FUNCTION setOutInt : INT
VAR_INPUT
	bol_GlobalEnableForce: BOOL;
	p_Output: POINTER TO T_Ctrl_IoInt;
END_VAR

// Copy real values
p_Output^.state := p_Output^.intern;

IF (p_Output^.EnForce AND bol_GlobalEnableForce) THEN
	p_Output^.map := p_Output^.force;
ELSE
	p_Output^.map := p_Output^.intern;
END_IF;

setOutInt := p_Output^.map;

END_FUNCTION

(* stored: Version 1.1.0.1, ProductVersion 3.1.0.18
   POU setOutInt: Id {e9ef2697-df64-4566-be18-d30e900ebf53} *)
